// TIA Portal V17 export
// export: Created 2026-04-13T11:12:42.0824964Z, ExportSetting WithDefaults, DisplayName Totally Integrated Automation Portal, DisplayVersion V17 Update 4, DisplayName TIA Portal Openness, DisplayVersion V17 Update 4, DisplayName TIA Portal Version Control Interface, DisplayVersion V17, DisplayName SINAMICS Startdrive Advanced, DisplayVersion V17, DisplayName SINAMICS Startdrive G130, G150, S120, S150, SINAMICS MV, S210, DisplayVersion V17, DisplayName SINAMICS Startdrive G110M, G120, G120C, G120D, G120P, G115D, DisplayVersion V17, DisplayName STEP 7 Professional, DisplayVersion V17 Update 4, DisplayName STEP 7 Safety, DisplayVersion V17, DisplayName WinCC Professional, DisplayVersion V17 Update 4
FUNCTION_BLOCK "自保持模式"   // FB83, SCL
{ S7_Optimized_Access := 'TRUE' }
VERSION : 0.1
// stored: AutoNumber true, IsIECCheckEnabled false, IsRetainMemResEnabled false, MemoryReserve 100, SetENOAutomatically false, UDAEnableTagReadback false
   VAR
      dooropened : Bool;
      homed : Bool;
      selfcheckmeet : Bool;
      sb_start : Bool;
      sb_stop : Bool;
      light : Bool;
   END_VAR
BEGIN
   #selfcheckmeet := (#dooropened AND #homed) OR #selfcheckmeet;

   IF NOT #selfcheckmeet THEN
       RETURN;
   END_IF;

   #light := (#sb_start OR #light) AND NOT #sb_stop;
END_FUNCTION_BLOCK
